FUNCTION F_silu : lreal
VAR_INPUT
	x : LREAL;
END_VAR

IF x > 1E2 THEN
	F_silu := x;
ELSIF x < -1E2 THEN
	F_silu := 0;
ELSE
	F_silu := x / (1 + EXP(-x));
END_IF

END_FUNCTION

(* stored: Version 1.1.0.1, ProductVersion 3.1.4024.12
   POU F_silu: Id {776c6fa3-c0e3-465d-991a-a3924569a053}, SpecialFunc None *)
